// TIA Portal V19 export
DATA_BLOCK "Simulation_DB"   // DB7
// stored: InstanceOfName Simulation, InstanceOfType FB
"Simulation"
   // VAR
   //    LGF_Error : Array[1..10] of Bool;
   //    LGF_Status : Array[1..10] of Word;
   //    RetValReal : Real;
   // END_VAR
BEGIN
END_DATA_BLOCK
